FUNCTION_BLOCK LoopREPEAT (* Template for an empty basic function block *)
  (* Standard: 61499-2; Description: Copyright (c) 2019 Jan Holzweber This program and the accompanying materials are made available under the terms of the Eclipse Public License 2.0 which is available at https://www.eclipse.org/legal/epl-2.0/ SPDX-License-Identifier: EPL-2.0 *)
  (* Version 1.0, 2019-06-05, jholz *)
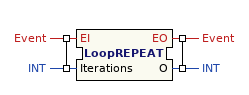
  EVENT_INPUT
    EI WITH Iterations;
  END_EVENT
  EVENT_OUTPUT
    EO WITH O;
  END_EVENT
  VAR_INPUT
    Iterations : INT;
  END_VAR
  VAR_OUTPUT
    O : INT;
  END_VAR
  VAR
    i : INT := 0; (* Internal Variable *)
  END_VAR
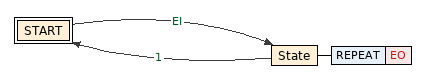
  EC_STATES
    START; (* Initial State *)
    State : REPEAT -> EO;
  END_STATES
  EC_TRANSITIONS
    START TO State := EI;
    State TO START := 1;
  END_TRANSITIONS
  ALGORITHM REPEAT IN ST: (* new algorithm *)
REPEAT
	O := O+i;
	i:= i+1;
UNTIL Iterations < i
END_REPEAT;
  END_ALGORITHM
END_FUNCTION_BLOCK
